Omron Sysmac Studio project MODBUS_TPC_CLIENT_NX1P2_LIBRARY_OPEN (Sysmac Studio 1.45.1.64010, StandardProject)

# Controller new_Controller_0: NX1P2-9024DT version 1.40
Units and slaves: Node86 : NX-ECC201 (E001); Unit 1 : NX-OD5121 (N1); Unit 2 : NX-OD4256 (N2); Unit 3 : NX-ID5342 (N3); Unit 4 : NX-ID5442 (N4); Node1 : GX-ID1611+OD16 (E002)
Task PrimaryTask (priority 4, period or condition 2000): Program0
Library OEN_Communication_V1_0_22 1.0.22 (contents left out)

VAR_GLOBAL
    NX1P2_OUT_0 : BOOL;  (* NX1P2_OUT *)
    NX1P2_OUT_1 : BOOL;  (* NX1P2_OUT *)
    NX1P2_OUT_2 : BOOL;  (* NX1P2_OUT *)
    NX1P2_OUT_3 : BOOL;  (* NX1P2_OUT *)
    NX1P2_OUT_4 : BOOL;  (* NX1P2_OUT *)
    NX1P2_OUT_5 : BOOL;  (* NX1P2_OUT *)
    NX1P2_OUT_6 : BOOL;  (* NX1P2_OUT *)
    NX1P2_OUT_7 : BOOL;  (* NX1P2_OUT *)
    NX1P2_OUT_8 : BOOL;  (* NX1P2_OUT *)
    NX1P2_OUT_9 : BOOL;  (* NX1P2_OUT *)
    GX_OUT_0 : BOOL;  (* OD_1611_DT; at ECAT://node#1/Write output 1st word/Out Bit00 *)
    GX_OUT_1 : BOOL;  (* OD_1611_DT; at ECAT://node#1/Write output 1st word/Out Bit01 *)
    GX_OUT_2 : BOOL;  (* OD_1611_DT; at ECAT://node#1/Write output 1st word/Out Bit02 *)
    GX_OUT_3 : BOOL;  (* OD_1611_DT; at ECAT://node#1/Write output 1st word/Out Bit03 *)
    GX_OUT_4 : BOOL;  (* OD_1611_DT; at ECAT://node#1/Write output 1st word/Out Bit04 *)
    GX_OUT_5 : BOOL;  (* OD_1611_DT; at ECAT://node#1/Write output 1st word/Out Bit05 *)
    GX_OUT_6 : BOOL;  (* OD_1611_DT; at ECAT://node#1/Write output 1st word/Out Bit06 *)
    GX_OUT_7 : BOOL;  (* OD_1611_DT; at ECAT://node#1/Write output 1st word/Out Bit07 *)
    GX_OUT_8 : BOOL;  (* OD_1611_DT; at ECAT://node#1/Write output 1st word/Out Bit08 *)
    GX_OUT_9 : BOOL;  (* OD_1611_DT; at ECAT://node#1/Write output 1st word/Out Bit09 *)
    GX_OUT_10 : BOOL;  (* OD_1611_DT; at ECAT://node#1/Write output 1st word/Out Bit10 *)
    GX_OUT_11 : BOOL;  (* OD_1611_DT; at ECAT://node#1/Write output 1st word/Out Bit11 *)
    GX_OUT_12 : BOOL;  (* OD_1611_DT; at ECAT://node#1/Write output 1st word/Out Bit12 *)
    GX_OUT_13 : BOOL;  (* OD_1611_DT; at ECAT://node#1/Write output 1st word/Out Bit13 *)
    GX_OUT_14 : BOOL;  (* OD_1611_DT; at ECAT://node#1/Write output 1st word/Out Bit14 *)
    GX_OUT_15 : BOOL;  (* OD_1611_DT; at ECAT://node#1/Write output 1st word/Out Bit15 *)
    REGISTER_GX_OUT : WORD;  (* OD_1611_DT; at ECAT://node#1/Write output 1st word *)
END_VAR

PROGRAM Program0
VAR
    DISCONNECT_TCP_CLIENT : BOOL;
    TCP_CLIENT_CONNECT : BOOL;
    T_CONNECT_TCP : TON;
    T_CONNECT_TCP_CLIENT : TON;
    MODBUS_CLIENT : OEN\Modbus\ModbusTCP_Client;
    REQUEST_CLIENT : ARRAY[0..1] OF OEN\Modbus\sModbusReq := [(Enable := True, NodeAdr := 0, FunctionCode := Fn03_ReadHoldingRegisters, Read := (StartAddressRemote := 0, StartAddressLocal := 0, Count := 4), Write := (StartAddressRemote := 0, StartAddressLocal := 0, Count := 0)), (Enable := True, NodeAdr := 0, FunctionCode := Fn16_WriteMultipleRegisters, Read := (StartAddressRemote := 0, StartAddressLocal := 0, Count := 0), Write := (StartAddressRemote := 4, StartAddressLocal := 4, Count := 6))];
    DATA_COIL_CLIENT : ARRAY[0..16] OF BOOL;
    DISCRETELINPUT_CLIENT : ARRAY[0..16] OF BOOL;
    INPUT_REGISTER_CLIENT : ARRAY[0..16] OF WORD;
    HOLDINGREGISTERR_CLIENT : ARRAY[0..16] OF WORD;
    REQUEST_DONE : BOOL;
    REQUEST_CLYCLE_TIME : TIME;
    TCP_CONNECT : BOOL;
    DATA_WRITE_0 : WORD;
    DATA_WRITE_1 : WORD;
    DATA_WRITE_2 : WORD;
END_VAR
VAR_EXTERNAL
    REGISTER_GX_OUT : WORD;
END_VAR

(* Section Section0: ladder, written here as Structured Text *)

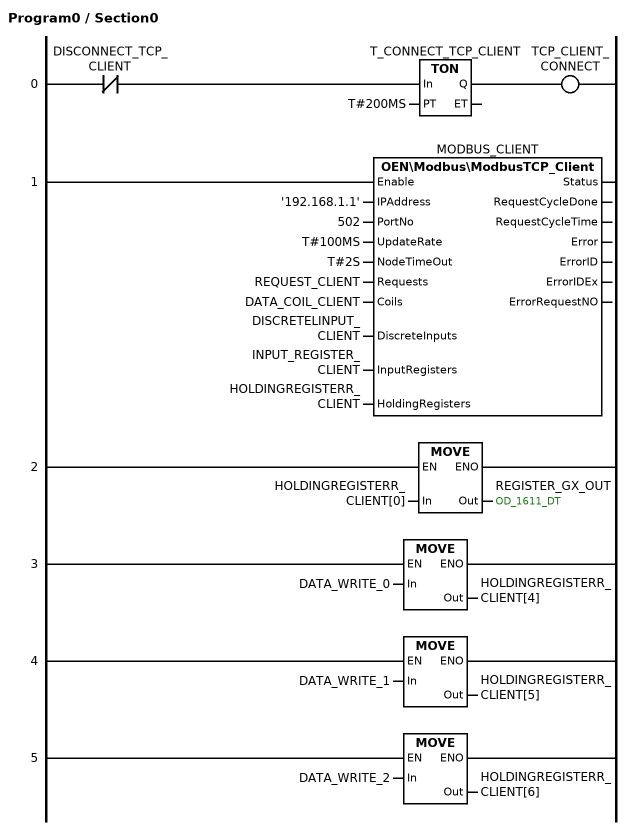
(* Rung 0 *)
T_CONNECT_TCP_CLIENT(In := NOT DISCONNECT_TCP_CLIENT, PT := T#200MS);
TCP_CLIENT_CONNECT := T_CONNECT_TCP_CLIENT.Q;
(* Rung 1 *)
MODBUS_CLIENT(Enable := TRUE, IPAddress := '192.168.1.1', PortNo := 502, UpdateRate := T#100MS, NodeTimeOut := T#2S, Requests := REQUEST_CLIENT, Coils := DATA_COIL_CLIENT, DiscreteInputs := DISCRETELINPUT_CLIENT, InputRegisters := INPUT_REGISTER_CLIENT, HoldingRegisters := HOLDINGREGISTERR_CLIENT);
(* Rung 2 *)
REGISTER_GX_OUT := HOLDINGREGISTERR_CLIENT[0];
(* Rung 3 *)
HOLDINGREGISTERR_CLIENT[4] := DATA_WRITE_0;
(* Rung 4 *)
HOLDINGREGISTERR_CLIENT[5] := DATA_WRITE_1;
(* Rung 5 *)
HOLDINGREGISTERR_CLIENT[6] := DATA_WRITE_2;
END_PROGRAM